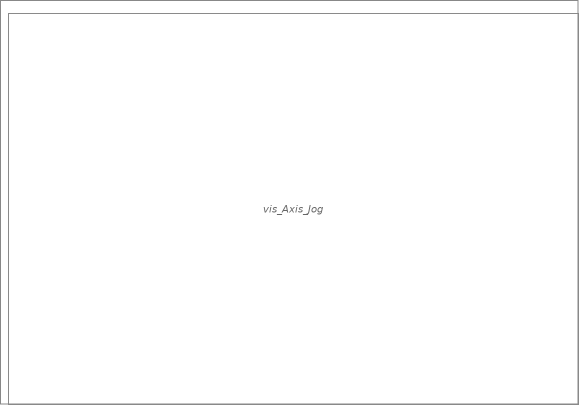
VISUALIZATION vis_Axis_Cont_Test  // 579x405
    Frame (8,13 571x392)
        shows vis_Axis_Jog(stAxis := stAxesfunctions[1])
END_VISUALIZATION

(* stored: Version 1.1.0.1, ProductVersion 3.1.4024.11
   Visu vis_Axis_Cont_Test: Id {ce49a78b-f127-4b0f-ab3e-7bac89d103a9} *)
